TYPE csp_transfer_infeed_waterfall_belt_status_enum :(
	CSP_TRANSFER_INFEED_WATERFALL_BELT_STATUS_NOT_INITIALIZED 							:= 0,
	CSP_TRANSFER_INFEED_WATERFALL_BELT_STATUS_DISABLED 									:= 10,
	CSP_TRANSFER_INFEED_WATERFALL_BELT_STATUS_ENABLE_REQUEST 								:= 70,
	CSP_TRANSFER_INFEED_WATERFALL_BELT_STATUS_ENABLING 									:= 80,
	CSP_TRANSFER_INFEED_WATERFALL_BELT_STATUS_ENABLED 									:= 100,
	CSP_TRANSFER_INFEED_WATERFALL_BELT_STATUS_RUNNING										:= 110,
	CSP_TRANSFER_INFEED_WATERFALL_BELT_STATUS_STOP_REQUEST 								:= 500,
	CSP_TRANSFER_INFEED_WATERFALL_BELT_STATUS_DISABLE_REQUEST 							:= 530,
	CSP_TRANSFER_INFEED_WATERFALL_BELT_STATUS_DISABLING 									:= 540
	) := CSP_TRANSFER_INFEED_WATERFALL_BELT_STATUS_NOT_INITIALIZED;
END_TYPE

(* stored: Version 1.1.0.1, ProductVersion 3.1.4022.12
   DUT csp_transfer_infeed_waterfall_belt_status_enum: Id {73f47ceb-27e5-450e-a52b-b08b011e2123} *)
